PROGRAM HeatCounter
VAR
	test_output : REAL;
	
	//cycle counter
	HeatCounter_CycleCount : UDINT;
    info  : GETCURTASKINDEX;
END_VAR

//test output for checking variable exchange between tasks with different cycle time
test_output := 1;
info();
HeatCounter_CycleCount := _TaskInfo[info.index].CycleCount;

END_PROGRAM

(* stored: Version 1.1.0.1, ProductVersion 3.1.4024.10
   POU HeatCounter: Id {4204b3f6-5c13-42c2-93aa-e47631f91a16}, SpecialFunc None *)
